FUNCTION_BLOCK ADI_SPLIT_9_UNGATED (* Wie ADI_SPLIT_9, aber OHNE Aenderungserkennung - reicht JEDES eingehende Event bedingungslos an alle 9 Ausgaenge weiter (fuer Verbraucher, die eine periodische Kadenz unabhaengig von Wertaenderung brauchen, z.B. Ableitungs-/Frequenzberechnungen). *)
  (* Standard: 61499-2; Description: Copyright (c) 2026 Meisterschulen am Ostbahnhof This program and the accompanying materials are made available under the terms of the Eclipse Public License 2.0 which is available at https://www.eclipse.org/legal/epl-2.0/ SPDX-License-Identifier: EPL-2.0 *)
  (* Version 1.0, 2026-08-31, Franz Höpfinger, Meisterschulen am Ostbahnhof *)
  PACKAGE adapter::events::unidirectional;
  IMPORT eclipse4diac::core::GenericClassName;
  {SET_ATTRIBUTE(eclipse4diac::core::GenericClassName, 'GEN_ADI_SPLIT')}
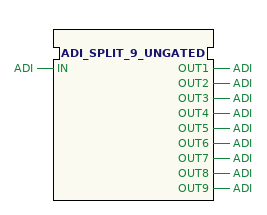
  SOCKETS
    IN : adapter::types::unidirectional::ADI;
  END_SOCKETS
  PLUGS
    OUT1 : adapter::types::unidirectional::ADI;
    OUT2 : adapter::types::unidirectional::ADI;
    OUT3 : adapter::types::unidirectional::ADI;
    OUT4 : adapter::types::unidirectional::ADI;
    OUT5 : adapter::types::unidirectional::ADI;
    OUT6 : adapter::types::unidirectional::ADI;
    OUT7 : adapter::types::unidirectional::ADI;
    OUT8 : adapter::types::unidirectional::ADI;
    OUT9 : adapter::types::unidirectional::ADI;
  END_PLUGS
END_FUNCTION_BLOCK
